// TwinCAT 3 PLC project Main
// ProgramVersion: 3.1.4024.0
// libraries:
//   Tc2_Standard, * (Beckhoff Automation GmbH)
//   Tc2_System, * (Beckhoff Automation GmbH)
//   Tc2_Utilities, * (Beckhoff Automation GmbH)
//   Tc3_JsonXml, * (Beckhoff Automation GmbH)
//   Tc3_Module, * (Beckhoff Automation GmbH)
//   TcUnit, * (www.tcunit.org)
//   mobject-core,0.7.0,mobject
//   mobject-server,0.17.0,mobject
// project tree:
//   / Param.TcGVL (not stored), PlcTask.TcTTO
//   POUs/ MAIN.TcPOU (not stored)
//   Tests/Mocks/ AdjustableSizeReplyRpcHandler.TcPOU, RejectWithMessageSyncHandler.TcPOU (not stored), SyncToAsyncEchoRpcHandler.TcPOU (not stored), RejectWithMessageAsyncHandler.TcPOU (not stored)
//   Tests/ Server_IntegrationTestSuite.TcPOU
//   Tests/_Internal/ ChunkedRequestData_TestSuite.TcPOU (not stored)
// real-time tasks:
//   TASK PlcTask: cycle T#10ms, priority 20, ADS port 350

CONFIGURATION Main
    RESOURCE PLC ON TwinCAT3
        TASK PlcTask(INTERVAL := T#10ms, PRIORITY := 20);
        PROGRAM MAIN WITH PlcTask : MAIN;
    END_RESOURCE
END_CONFIGURATION

// ---- Tests/Mocks/AdjustableSizeReplyRpcHandler.TcPOU
FUNCTION_BLOCK AdjustableSizeReplyRpcHandler IMPLEMENTS I_SynchronousRpcHandler
VAR
END_VAR

METHOD Handle
VAR_INPUT
	Parameters : I_Deserializer;
	Response : I_SynchronousRpcResponse;
END_VAR
VAR
	deserializerFeedback : DeserializerFeedback;
	size : UDINT;
	pBytes : POINTER TO BYTE;
	currentPos : POINTER TO BYTE;
	i : UDINT;
	count : BYTE;
END_VAR
IF NOT Parameters.TryGetKeyUdint('Size', size, deserializerFeedback) THEN
	Response.RejectWithMessage('Missing Size parameter');
	RETURN;
END_IF

IF size = 0 THEN 
	Response.CompleteWithNull();
END_IF

pBytes := __NEW(BYTE, size);
FOR i := 0 TO size -1 DO
	currentPos := pBytes + i;
	currentPos^ := count;
	count := count + 1;
END_FOR

Response.CompleteWithBytesAsHex(pBytes, UDINT_TO_DINT(size));

__Delete(pBytes);
END_METHOD

END_FUNCTION_BLOCK

// ---- Tests/Server_IntegrationTestSuite.TcPOU
FUNCTION_BLOCK Server_IntegrationTestSuite EXTENDS TcUnit.FB_TestSuite
VAR
	// variables for TestAsyncEchoRpcCallAndResponse
	testAsyncEchoRpcCallAndResponseSetup : BOOL;
	testAsyncEchoRpcCallAndResponseServer : RpcServer;
	testAsyncEchoRpcCallAndResponseAsyncEchoRpcHandler : SyncToAsyncEchoRpcHandler;
	testAsyncEchoRpcCallAndResponseOutput : ResponseData;
	
	// variables for TestConcatRpcCallAndResponse
	testConcatRpcCallAndResponseOutput : ResponseData;
	
	// variables for TestAsyncConcatRpcCallAndResponse
	testAsyncConcatRpcCallAndResponseOutput : ResponseData;
	
	// variables for TestAsyncRejectMessage
	testAsyncRejectMessageOutput : ResponseData;
	
	// variables for TestSyncRejectMessage
	testSyncRejectMessageOutput : ResponseData;
	
END_VAR

TestSyncToAsyncEchoRpcCallAndResponse();
TestConcatRpcCallAndResponse();
TestConcatRpcCallAndResponseWithChunkedRequest();
TestAsyncConcatRpcCallAndResponse();
TestAsyncRejectMessage();
TestSyncRejectMessage();

METHOD TestAsyncConcatRpcCallAndResponse
VAR
	server : RpcServer;
	asyncConcatStringRpcHandler : AsyncConcatStringRpcHandler;
	header : T_MAXSTRING := '{"Type":"RPC 1.0","Method-Name":"concat","Content-Type":"application/json"}';
    payload : T_MAXSTRING := '{"STR1":"hello", "STR2":"world"}';
	followupHeader : T_MAXSTRING := '{"Type":"RPC 1.0","Accept":"application/json","Method-Name":"asyncEcho","Response-Id":"1","Session-Id":"1"}';
	followupPayload : T_MAXSTRING := '';
	expected : T_MAXSTRING := '"helloworld"';
	actual : T_MAXSTRING;
END_VAR
TEST('TestAsyncConcatRpcCallAndResponse');

server.RegisterAsynchronousRpcHandler('concat',asyncConcatStringRpcHandler);

testAsyncConcatRpcCallAndResponseOutput := server.HandleRequest(header,payload);
server.CyclicCall();
testAsyncConcatRpcCallAndResponseOutput := server.HandleRequest(followupHeader, followupPayload);
actual := testAsyncConcatRpcCallAndResponseOutput.Payload;

AssertEquals(
	Expected := expected, 
	Actual := actual,
	Message := 'Did not produce the expected result'
);

TEST_FINISHED();
END_METHOD

METHOD TestAsyncRejectMessage
VAR
	server : RpcServer;
	rejectWithMessageAsyncHandler : RejectWithMessageAsyncHandler;
	header : T_MAXSTRING := '{"Type":"RPC 1.0","Method-Name":"reject","Content-Type":"application/json"}';
    payload : T_MAXSTRING := '';
	followupHeader : T_MAXSTRING := '{"Response-Id":"1","Session-Id":"1"}';
	followupPayload : T_MAXSTRING := '';
	expectedFirstReply : T_MAXSTRING := '{"Session-Id":"1","Status":"Pending","Response-Id":"1"}';
	expectedSecondReply : T_MAXSTRING := '{"Session-Id":"1","Status":"Error","Message":"This is the reject message"}';
	actual : T_MAXSTRING;
END_VAR
TEST('TestAsyncRejectMessage');

server.RegisterAsynchronousRpcHandler('reject',rejectWithMessageAsyncHandler);

testAsyncRejectMessageOutput := server.HandleRequest(header,payload);
actual := testAsyncRejectMessageOutput.Header;

AssertEquals(
	Expected := expectedFirstReply, 
	Actual := actual,
	Message := 'Did not reply that the request was being processed'
);

server.CyclicCall();


testAsyncRejectMessageOutput := server.HandleRequest(followupHeader,followupPayload);
actual := testAsyncRejectMessageOutput.Header;


AssertEquals(
	Expected := expectedSecondReply, 
	Actual := actual,
	Message := 'Did not produce the expected result'
);

TEST_FINISHED();
END_METHOD

METHOD TestConcatRpcCallAndResponse
VAR
	server : RpcServer;
	concatStringRpcHandler : ConcatStringRpcHandler;
	header : T_MAXSTRING := '{"Type":"RPC 1.0","Method-Name":"concat","Content-Type":"application/json"}';
    payload : T_MAXSTRING := '{"STR1":"hello", "STR2":"world"}';
	expected : T_MAXSTRING := '"helloworld"';
	actual : T_MAXSTRING;
END_VAR
TEST('TestConcatRpcCallAndResponse');

server.RegisterSynchronousRpcHandler('concat',concatStringRpcHandler);

testConcatRpcCallAndResponseOutput := server.HandleRequest(header,payload);
actual := testConcatRpcCallAndResponseOutput.Payload;

AssertEquals(
	Expected := expected, 
	Actual := actual,
	Message := 'Did not produce the expected result'
);

TEST_FINISHED();
END_METHOD

METHOD TestConcatRpcCallAndResponseWithChunkedRequest
VAR
	server : RpcServer;
	concatStringRpcHandler : ConcatStringRpcHandler;
	chunk1Header : T_MAXSTRING := '{"Type":"RPC 1.0","Method-Name":"concat","Request-Id":"abc","Has-More-Chunks":true, "Chunk-Sequence":1, "Chunk-Total":2, "Content-Type":"application/json"}';
    chunk1payload : T_MAXSTRING := '{"STR1":"hello",';
	chunk2Header : T_MAXSTRING := '{"Type":"RPC 1.0","Session-Id":"1","Method-Name":"concat","Request-Id":"abc","Has-More-Chunks":false, "Chunk-Sequence":2, "Chunk-Total":2, "Content-Type":"application/json"}';
    chunk2payload : T_MAXSTRING := ' "STR2":"world"}';
	expected : T_MAXSTRING := '"helloworld"';
	out : ResponseData;
END_VAR
//TEST('TestConcatRpcCallAndResponseWithChunkedRequest');

//server.RegisterRpcHandler('concat',concatStringRpcHandler);

//out := server.HandleRequest(chunk1Header,chunk1payload);
//out := server.HandleRequest(chunk2Header,chunk2payload);

//AssertTrue(
//	Condition := expected = out.Payload,
//	Message := 'Did not produce the expected result'
//);

//TEST_FINISHED();
END_METHOD

METHOD TestSyncRejectMessage
VAR
	server : RpcServer;
	rejectWithMessageSyncHandler : RejectWithMessageSyncHandler;
	header : T_MAXSTRING := '{"Type":"RPC 1.0","Method-Name":"reject","Content-Type":"application/json"}';
    payload : T_MAXSTRING := '';
	expected : T_MAXSTRING := '{"Session-Id":"1","Status":"Error","Message":"This is the reject message"}';
	actual : T_MAXSTRING;
END_VAR
TEST('TestSyncRejectMessage');

server.RegisterSynchronousRpcHandler('reject',rejectWithMessageSyncHandler);

testSyncRejectMessageOutput := server.HandleRequest(header,payload);
actual := testAsyncRejectMessageOutput.Header;

AssertEquals(
	Expected := expected, 
	Actual := actual,
	Message := 'Did not produce the expected result'
);

TEST_FINISHED();
END_METHOD

METHOD TestSyncToAsyncEchoRpcCallAndResponse
VAR
	header : T_MAXSTRING := '{"Type":"RPC 1.0","Accept":"application/json","Method-Name":"asyncEcho","Content-Type":"application/json"}';
    payload : T_MAXSTRING := '{"Echo":"hello"}';
	followupHeader : T_MAXSTRING := '{"Type":"RPC 1.0","Accept":"application/json","Method-Name":"asyncEcho","Response-Id":"1","Session-Id":"1"}';
	followuPayload : T_MAXSTRING := '{"Echo":"hello"}';
	expected : T_MAXSTRING := '"hello"';
	actual : T_MAXSTRING;
END_VAR
TEST('TestAsyncEchoRpcCallAndResponse');

IF NOT testAsyncEchoRpcCallAndResponseSetup THEN
	testAsyncEchoRpcCallAndResponseServer.RegisterSynchronousRpcHandler('asyncEcho',testAsyncEchoRpcCallAndResponseAsyncEchoRpcHandler);
	testAsyncEchoRpcCallAndResponseOutput := testAsyncEchoRpcCallAndResponseServer.HandleRequest(header,payload);
	testAsyncEchoRpcCallAndResponseSetup := TRUE;	
END_IF

testAsyncEchoRpcCallAndResponseAsyncEchoRpcHandler.CyclicCall();

IF testAsyncEchoRpcCallAndResponseAsyncEchoRpcHandler.Busy THEN
	RETURN;
END_IF

testAsyncEchoRpcCallAndResponseOutput := testAsyncEchoRpcCallAndResponseServer.HandleRequest(followupHeader,followuPayload);
actual := testAsyncEchoRpcCallAndResponseOutput.Payload;

AssertEquals(
	Expected := expected, 
	Actual := actual,
	Message := 'Did not produce the expected result'
);

TEST_FINISHED();
END_METHOD

END_FUNCTION_BLOCK
